INTERFACE I_Blank EXTENDS __SYSTEM.IQueryInterface

END_INTERFACE

(* stored: Version 1.1.0.1, ProductVersion 3.1.4024.12
   Itf I_Blank: Id {aaf61729-6beb-46e2-a224-9cdd9e42e530} *)
